// Block: PPrgArchive7

DATA_BLOCK PPrgArchive7
VERSION : 0.1
   NON_RETAIN
   VAR
      PRG : Array[601..700] of PPrg_Data;
   END_VAR

BEGIN
   // No initialization required
END_DATA_BLOCK
